FUNCTION_BLOCK RED_LIGHT (* lamp *)
  (* Standard: 61499-2 *)
  (* Version 03-07-12, GASR *)
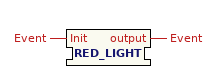
  EVENT_INPUT
    Init;
  END_EVENT
  EVENT_OUTPUT
    output;
  END_EVENT
  SERVICE RED_LIGHT/LIGHT_SIM
    SEQUENCE seq1
      RED_LIGHT.Init() -> LIGHT_SIM.on();
    END_SEQUENCE
  END_SERVICE
END_FUNCTION_BLOCK
